// TIA Portal V20 export
TYPE "typeSequenceControlNodeJobInterface_topTapeFixStage"
// stored: Namespace Unit1.Em3
   STRUCT
      loadJob2 : "LER_typeJobInterface";
      taping1Job3 : "LER_typeJobInterface";
      taping2Job4 : "LER_typeJobInterface";
      unloadJob5 : "LER_typeJobInterface";
   END_STRUCT;
END_TYPE
